{attribute 'enable_dynamic_creation'}
FUNCTION_BLOCK FutureMCPower EXTENDS FB_AbstructFuture
VAR_INPUT
END_VAR
VAR_OUTPUT
END_VAR
VAR
	_axis: REFERENCE TO AXIS_REF;
	_override: LREAL := 100.0;
	_enable_positive:	BOOL := TRUE; 
	_enable_negative:	BOOL := TRUE;
	_fb_power	: MC_Power;
	_mc_reset	: MC_Reset;
	_option : ST_PowerOptions;
	_buffer_mode : MC_BufferMode;
	_error_id :UDINT;
END_VAR

METHOD abort : BOOL // Return TRUE if finish.
_fb_power(
	Axis:= _axis, 
	Enable:= FALSE, 
	Enable_Positive:= FALSE, 
	Enable_Negative:= FALSE, 
	Override:= _override, 
	BufferMode:= _buffer_mode, 
	Options:= _option, 
);	

abort := NOT _fb_power.Status;
END_METHOD

METHOD error_reset : BOOL // Must be overrided if future has any errors.
VAR_INST
	_exec_state : UDINT;
END_VAR
IF _error_id <> 0 THEN
	CASE _exec_state OF
		0:
			_mc_reset(Axis := _axis, Execute := FALSE);
			_mc_reset(Axis:= _axis, Execute := TRUE );
			_exec_state := 1;
		1:
			IF _mc_reset.Busy THEN
				_mc_reset(Axis:= _axis,Execute := FALSE);
			END_IF
	END_CASE
	
	_error_id := _mc_reset.ErrorID;
	error_reset := _mc_reset.Done;
ELSE
	error_reset := TRUE;
END_IF
END_METHOD

METHOD execute : BOOL // Return TRUE if finish.

_fb_power(
	Axis:= _axis, 
	Enable:= TRUE, 
	Enable_Positive:= _enable_positive, 
	Enable_Negative:= _enable_negative, 
	Override:= _override, 
	BufferMode:= _buffer_mode, 
	Options:= _option, 
);

_error_id := _fb_power.ErrorID;
execute := NOT _fb_Power.Status;
END_METHOD

PROPERTY nErrorID : UDINT
GET
nErrorID := _error_id;
END_GET
SET
END_SET
END_PROPERTY

METHOD set_options : BOOL
VAR_INPUT
	Enable_Positive:	BOOL; 
	Enable_Negative:	BOOL;
	Override:			LREAL := 100;
	buffer_mode : MC_BufferMode;
	option : ST_PowerOptions;
END_VAR
_override := Override;
_enable_positive := Enable_Positive;
_enable_negative := Enable_Negative;
_buffer_mode := buffer_mode;
_option := option;
END_METHOD

METHOD set_parameters : BOOL
VAR_INPUT
	axis : REFERENCE TO AXIS_REF;
END_VAR
_axis REF= axis;
END_METHOD

END_FUNCTION_BLOCK

(* stored: Version 1.1.0.1, ProductVersion 3.1.4024.12
   POU FutureMCPower: Id {53bbc5ad-8cba-4d76-9354-ff6510473cd2}, SpecialFunc None
   Method abort: Id {a2ebf70c-c955-4d49-84ab-bdec62d66a45}
   Method error_reset: Id {fbfcfc82-515e-4f7c-ae99-279462150b8a}
   Method execute: Id {f127afa9-edb6-44ee-8a9c-b074dfb931e5}
   Property nErrorID: Id {c3c180c4-d69e-4a51-9c5f-b279b0d62fc4}
   Get Get: Id {8d5bdd1d-5bd8-4346-a4c9-03a10b43c4fe}
   Set Set: Id {9e9054ff-5773-4183-aecd-61fc3fb4858d}
   Method set_options: Id {93406fea-fe89-4d4b-b9dc-dafbd821cdd6}
   Method set_parameters: Id {c4fee9f1-f0d8-457c-bc4c-46597f9f2a6d} *)
